(* PLC project Sin nombre, Desconocido Sin nombre 1 *)
(* stored: creationDateTime 2025-10-12T14:16:42, modificationDateTime 2025-10-24T16:56:18 *)

PROGRAM elnuestro
  VAR
    Fotorresistor AT %IW0 : UINT;
    Pot AT %IW1 : UINT;
    Sensor_inc AT %IX0.1 : BOOL;
    led_inc AT %QX0.1 : BOOL;
    altavoz AT %QX0.0 : BOOL;
    laser AT %QW1 : UINT;
  END_VAR
  VAR
    ritmo_alarma_inc : TP;
    ritmo_alarma_inc_2 : TOF;
    duracion_alarma_laser : TP;
    ritmo_alarma_laser : TP;
    ritmo_alarma_laser_2 : TOF;
  END_VAR
  VAR  (* added by the conversion: wires and edge detectors of the diagram *)
    _AND13_OUT : BOOL;
    _GE8_OUT : BOOL;
  END_VAR

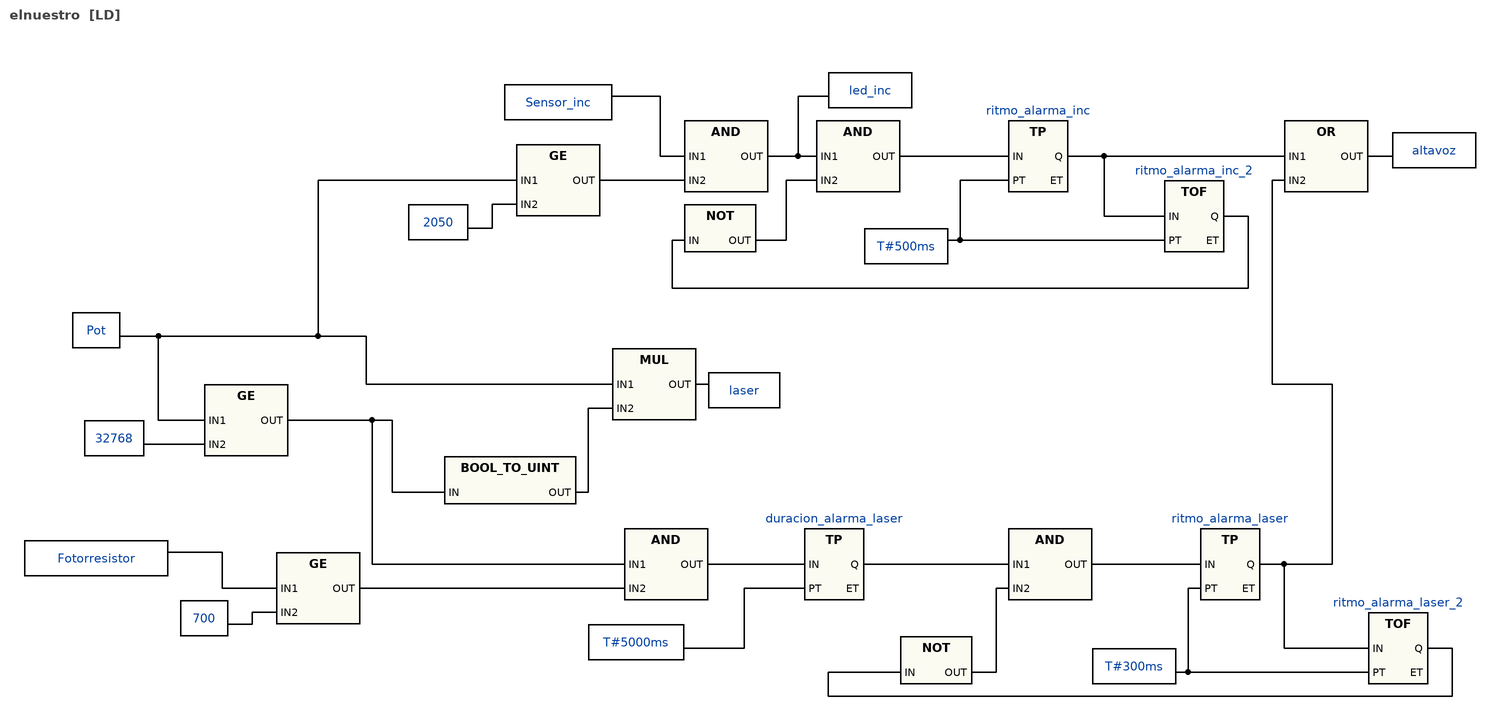
(* LD diagram, written out as Structured Text *)
_AND13_OUT := Sensor_inc AND Pot >= 2050;
ritmo_alarma_inc_2(IN := ritmo_alarma_inc.Q, PT := T#500ms);
ritmo_alarma_inc(IN := _AND13_OUT AND NOT ritmo_alarma_inc_2.Q, PT := T#500ms);
_GE8_OUT := Pot >= 32768;
duracion_alarma_laser(IN := _GE8_OUT AND Fotorresistor >= 700, PT := T#5000ms);
ritmo_alarma_laser_2(IN := ritmo_alarma_laser.Q, PT := T#300ms);
ritmo_alarma_laser(IN := duracion_alarma_laser.Q AND NOT ritmo_alarma_laser_2.Q, PT := T#300ms);
altavoz := ritmo_alarma_inc.Q OR ritmo_alarma_laser.Q;
laser := Pot * BOOL_TO_UINT(_GE8_OUT);
led_inc := _AND13_OUT;
END_PROGRAM

CONFIGURATION Config0
  RESOURCE Res0 ON PLC
    TASK task0(INTERVAL := T#20ms, PRIORITY := 0);
    PROGRAM instance0 WITH task0 : elnuestro;
  END_RESOURCE
END_CONFIGURATION
